Fanuc TP program (LS listing): START_BLOW.LS

/PROG  START_BLOW	  Macro
/ATTR
OWNER		= MNEDITOR;
COMMENT		= "";
PROG_SIZE	= 146;
CREATE		= DATE 25-07-07  TIME 19:33:10;
MODIFIED	= DATE 25-07-07  TIME 19:33:10;
FILE_NAME	= ;
VERSION		= 0;
LINE_COUNT	= 1;
MEMORY_SIZE	= 514;
PROTECT		= READ_WRITE;
TCD:  STACK_SIZE	= 0,
      TASK_PRIORITY	= 50,
      TIME_SLICE	= 0,
      BUSY_LAMP_OFF	= 0,
      ABORT_REQUEST	= 0,
      PAUSE_REQUEST	= 0;
DEFAULT_GROUP	= *,*,*,*,*;
CONTROL_CODE	= 00000000 00000000;
/MN
   1:  DO[7:OFF:blow]=ON ;
/POS
/END
